FUNCTION_BLOCK CmdWaterDischargeSLB_HMI (* Service Interface Function Block Type *)
  (* Standard: 61499-2 *)
  (* Version 1.0, 9/30/2026, Claude/Hidryco, Schneider Electric, Rev1 - Parametros Cmax/C2/C3/T_C2/T_C3 e T_Restart/T_FlowLL (persistentes) *)
  PACKAGE SE.Nereda;
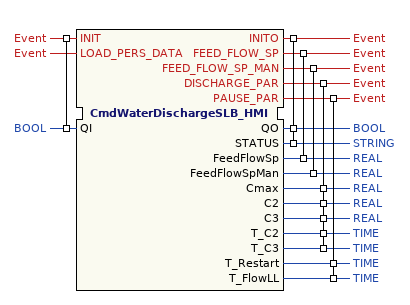
  EVENT_INPUT
    INIT WITH QI;
    LOAD_PERS_DATA;
  END_EVENT
  EVENT_OUTPUT
    INITO WITH QO, STATUS;
    FEED_FLOW_SP WITH FeedFlowSp;
    FEED_FLOW_SP_MAN WITH FeedFlowSpMan;
    DISCHARGE_PAR WITH Cmax, C2, C3, T_C2, T_C3; (* Parametros das bombas de sobrenadante *)
    PAUSE_PAR WITH T_Restart, T_FlowLL; (* Parametros da pausa da descarga de sobrenadante *)
  END_EVENT
  VAR_INPUT
    QI : BOOL;
  END_VAR
  VAR_OUTPUT
    QO : BOOL; (* Event Output Qualifier *)
    STATUS : STRING; (* Service Status *)
    FeedFlowSp : REAL;
    FeedFlowSpMan : REAL;
    Cmax : REAL; (* Vazao maxima de 1 bomba [m3/h] - acima dela entra a 2a bomba *)
    C2 : REAL; (* Vazao por bomba na entrada da 2a bomba [m3/h] *)
    C3 : REAL; (* Vazao por bomba abaixo da qual sai 1 bomba [m3/h] *)
    T_C2 : TIME; (* Tempo em C2 (reducao e aceleracao) *)
    T_C3 : TIME; (* Tempo abaixo de C3 para retirar 1 bomba *)
    T_Restart : TIME; (* Pausa: tempo para retomar apos a causa (nivel L / vazao LL) sair *)
    T_FlowLL : TIME; (* Vazao LL do 49FT0004 com bomba rodando por este tempo = pausa (0 = desabilitado) *)
  END_VAR
  SERVICE /
    SEQUENCE 
    END_SEQUENCE
  END_SERVICE
END_FUNCTION_BLOCK
